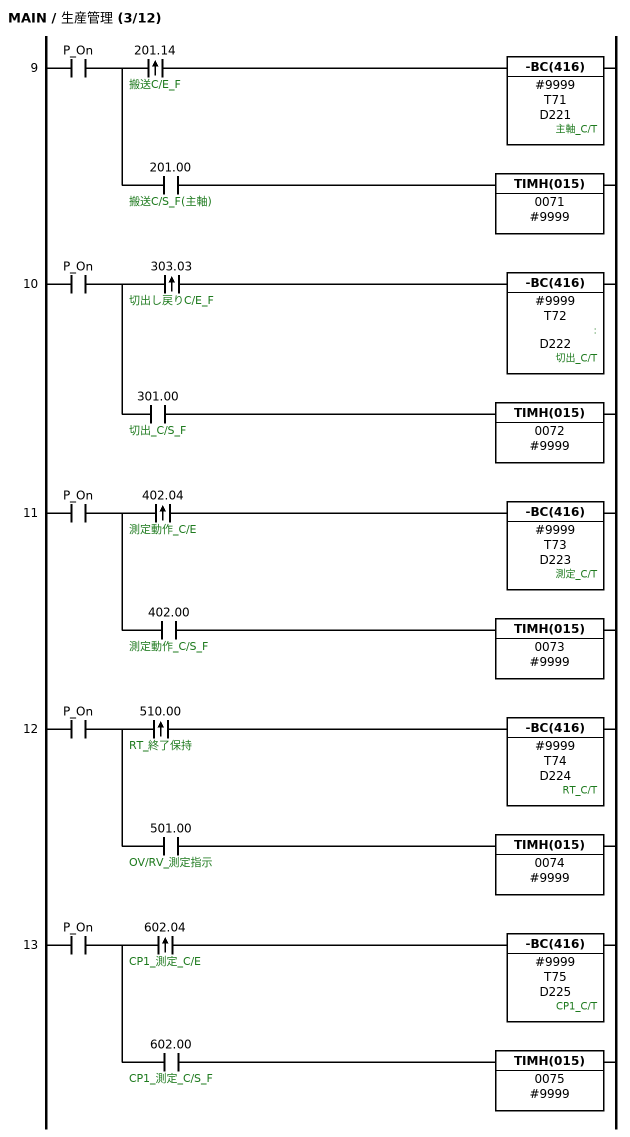
; [picture p24: MAIN / 生産管理, rungs 9-13]
; rung 9
LD P_On
OUT TR0
@AND 201.14  ; 搬送C/E_F
-BC(416) #9999 T71 D221  ; 主軸_C/T
LD TR0
AND 201.00  ; 搬送C/S_F(主軸)
TIMH(015) 0071 #9999
; rung 10
LD P_On
OUT TR0
@AND 303.03  ; 切出し戻りC/E_F
-BC(416) #9999 T72 D222  ; :, 切出_C/T
LD TR0
AND 301.00  ; 切出_C/S_F
TIMH(015) 0072 #9999
; rung 11
LD P_On
OUT TR0
@AND 402.04  ; 測定動作_C/E
-BC(416) #9999 T73 D223  ; 測定_C/T
LD TR0
AND 402.00  ; 測定動作_C/S_F
TIMH(015) 0073 #9999
; rung 12
LD P_On
OUT TR0
@AND 510.00  ; RT_終了保持
-BC(416) #9999 T74 D224  ; RT_C/T
LD TR0
AND 501.00  ; OV/RV_測定指示
TIMH(015) 0074 #9999
; rung 13
LD P_On
OUT TR0
@AND 602.04  ; CP1_測定_C/E
-BC(416) #9999 T75 D225  ; CP1_C/T
LD TR0
AND 602.00  ; CP1_測定_C/S_F
TIMH(015) 0075 #9999

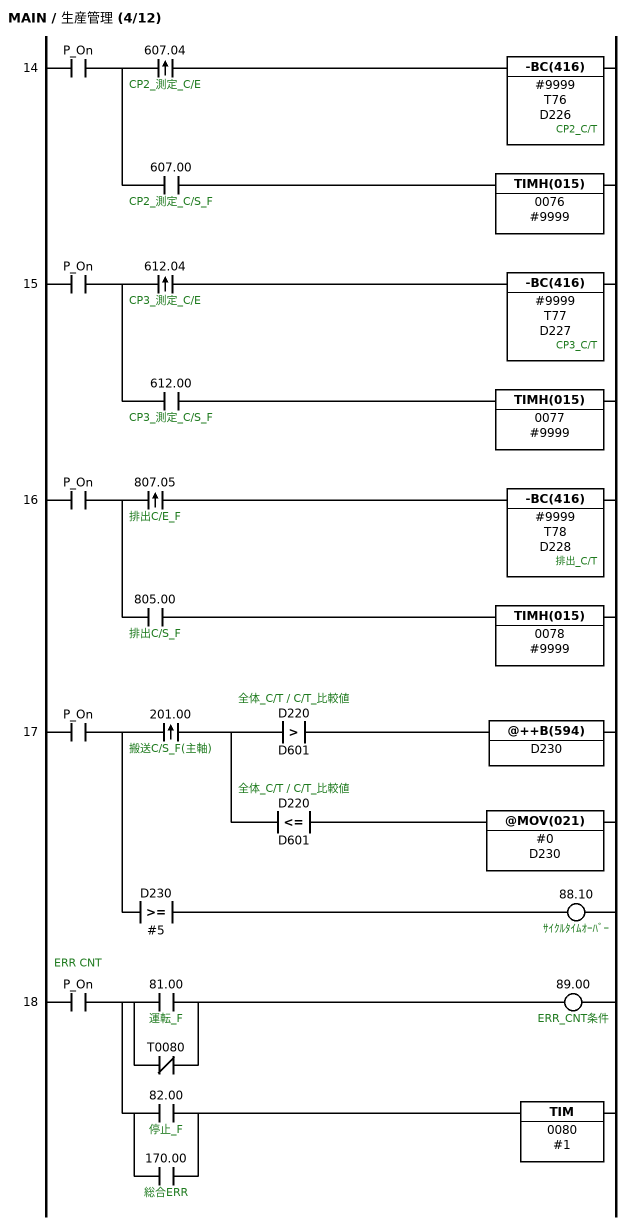
; rung 14
LD P_On
OUT TR0
@AND 607.04  ; CP2_測定_C/E
-BC(416) #9999 T76 D226  ; CP2_C/T
LD TR0
AND 607.00  ; CP2_測定_C/S_F
TIMH(015) 0076 #9999
; rung 15
LD P_On
OUT TR0
@AND 612.04  ; CP3_測定_C/E
-BC(416) #9999 T77 D227  ; CP3_C/T
LD TR0
AND 612.00  ; CP3_測定_C/S_F
TIMH(015) 0077 #9999
; rung 16
LD P_On
OUT TR0
@AND 807.05  ; 排出C/E_F
-BC(416) #9999 T78 D228  ; 排出_C/T
LD TR0
AND 805.00  ; 排出C/S_F
TIMH(015) 0078 #9999
; rung 17
LD P_On
OUT TR0
@AND 201.00  ; 搬送C/S_F(主軸)
OUT TR1
AND>(320) D220 D601  ; 全体_C/T, C/T_比較値
@++B(594) D230
LD TR1
AND<=(315) D220 D601  ; 全体_C/T, C/T_比較値
@MOV(021) #0 D230
LD TR0
AND>=(325) D230 #5
OUT 88.10  ; ｻｲｸﾙﾀｲﾑｵｰﾊﾞｰ
; rung 18: ERR CNT
LD P_On
OUT TR0
LD 81.00  ; 運転_F
ORNOT T0080
ANDLD
OUT 89.00  ; ERR_CNT条件
LD TR0
LD 82.00  ; 停止_F
OR 170.00  ; 総合ERR
ANDLD
TIM 0080 #1

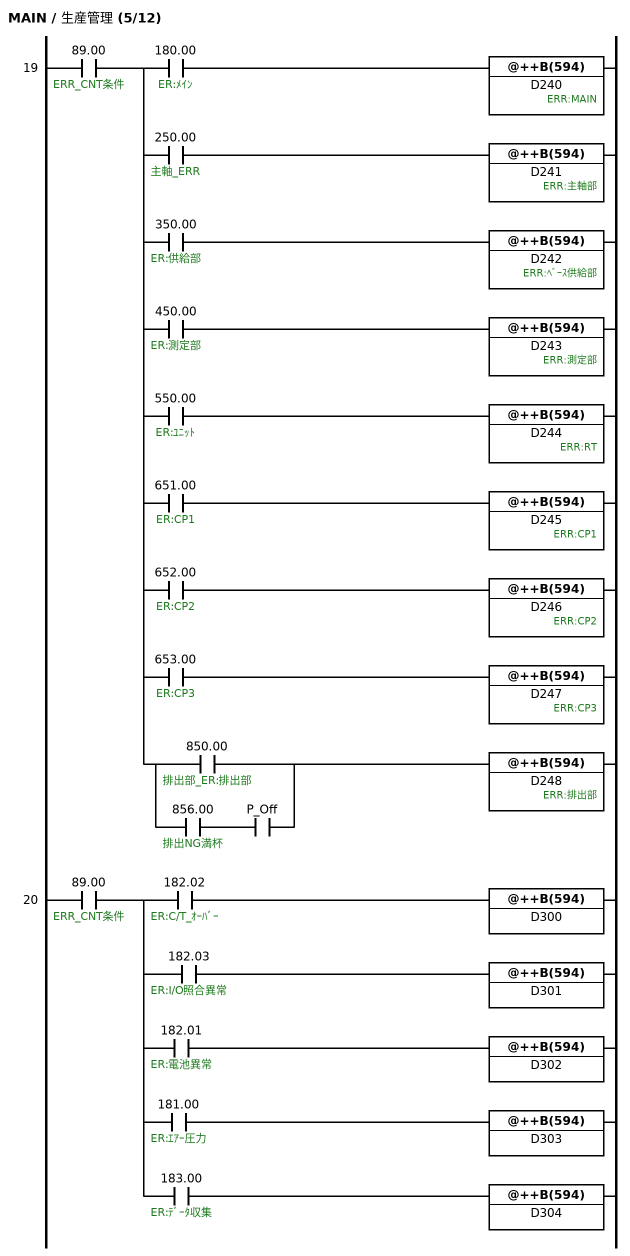
; rung 19
LD 89.00  ; ERR_CNT条件
OUT TR0
AND 180.00  ; ER:ﾒｲﾝ
@++B(594) D240  ; ERR:MAIN
LD TR0
AND 250.00  ; 主軸_ERR
@++B(594) D241  ; ERR:主軸部
LD TR0
AND 350.00  ; ER:供給部
@++B(594) D242  ; ERR:ﾍﾞｰｽ供給部
LD TR0
AND 450.00  ; ER:測定部
@++B(594) D243  ; ERR:測定部
LD TR0
AND 550.00  ; ER:ﾕﾆｯﾄ
@++B(594) D244  ; ERR:RT
LD TR0
AND 651.00  ; ER:CP1
@++B(594) D245  ; ERR:CP1
LD TR0
AND 652.00  ; ER:CP2
@++B(594) D246  ; ERR:CP2
LD TR0
AND 653.00  ; ER:CP3
@++B(594) D247  ; ERR:CP3
LD TR0
LD 850.00  ; 排出部_ER:排出部
LD 856.00  ; 排出NG満杯
AND P_Off
ORLD
ANDLD
@++B(594) D248  ; ERR:排出部
; rung 20
LD 89.00  ; ERR_CNT条件
OUT TR0
AND 182.02  ; ER:C/T_ｵｰﾊﾞｰ
@++B(594) D300
LD TR0
AND 182.03  ; ER:I/O照合異常
@++B(594) D301
LD TR0
AND 182.01  ; ER:電池異常
@++B(594) D302
LD TR0
AND 181.00  ; ER:ｴｱｰ圧力
@++B(594) D303
LD TR0
AND 183.00  ; ER:ﾃﾞｰﾀ収集
@++B(594) D304

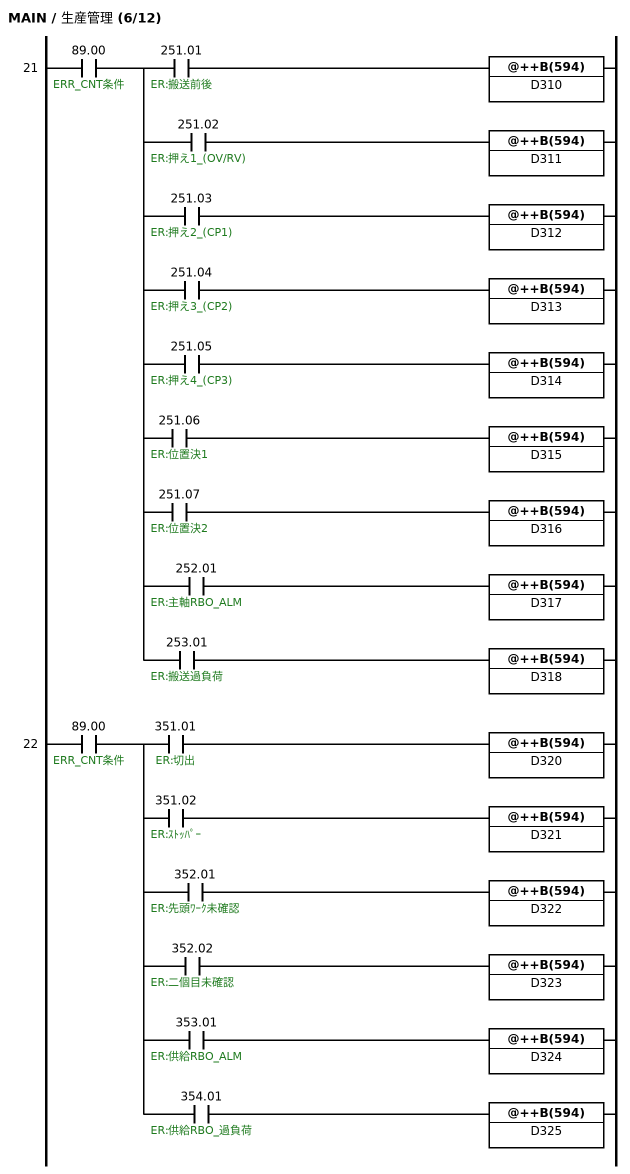
; rung 21
LD 89.00  ; ERR_CNT条件
OUT TR0
AND 251.01  ; ER:搬送前後
@++B(594) D310
LD TR0
AND 251.02  ; ER:押え1_(OV/RV)
@++B(594) D311
LD TR0
AND 251.03  ; ER:押え2_(CP1)
@++B(594) D312
LD TR0
AND 251.04  ; ER:押え3_(CP2)
@++B(594) D313
LD TR0
AND 251.05  ; ER:押え4_(CP3)
@++B(594) D314
LD TR0
AND 251.06  ; ER:位置決1
@++B(594) D315
LD TR0
AND 251.07  ; ER:位置決2
@++B(594) D316
LD TR0
AND 252.01  ; ER:主軸RBO_ALM
@++B(594) D317
LD TR0
AND 253.01  ; ER:搬送過負荷
@++B(594) D318
; rung 22
LD 89.00  ; ERR_CNT条件
OUT TR0
AND 351.01  ; ER:切出
@++B(594) D320
LD TR0
AND 351.02  ; ER:ｽﾄｯﾊﾟｰ
@++B(594) D321
LD TR0
AND 352.01  ; ER:先頭ﾜｰｸ未確認
@++B(594) D322
LD TR0
AND 352.02  ; ER:二個目未確認
@++B(594) D323
LD TR0
AND 353.01  ; ER:供給RBO_ALM
@++B(594) D324
LD TR0
AND 354.01  ; ER:供給RBO_過負荷
@++B(594) D325

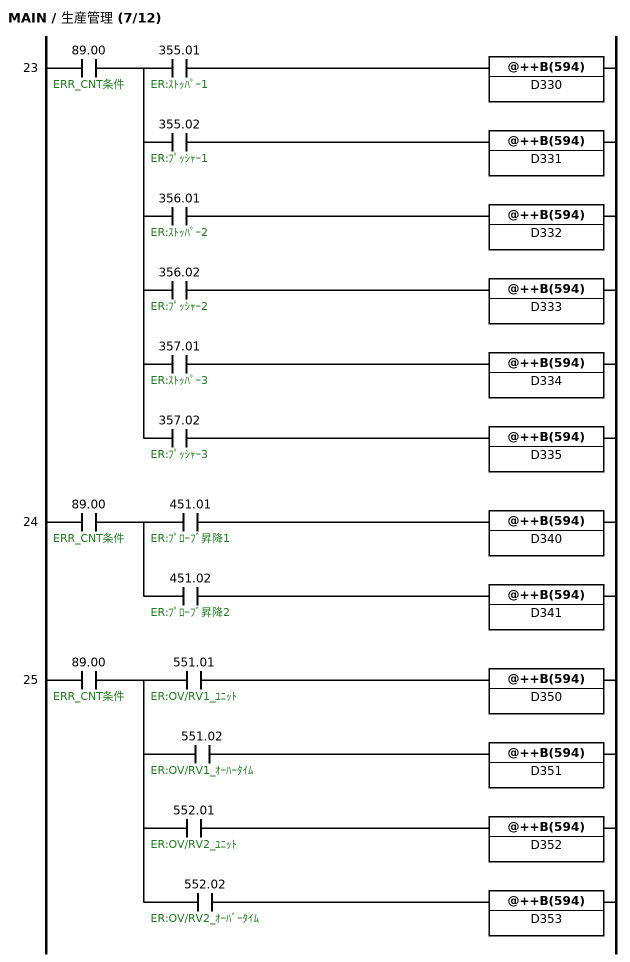
; rung 23
LD 89.00  ; ERR_CNT条件
OUT TR0
AND 355.01  ; ER:ｽﾄｯﾊﾟｰ1
@++B(594) D330
LD TR0
AND 355.02  ; ER:ﾌﾟｯｼｬｰ1
@++B(594) D331
LD TR0
AND 356.01  ; ER:ｽﾄｯﾊﾟｰ2
@++B(594) D332
LD TR0
AND 356.02  ; ER:ﾌﾟｯｼｬｰ2
@++B(594) D333
LD TR0
AND 357.01  ; ER:ｽﾄｯﾊﾟｰ3
@++B(594) D334
LD TR0
AND 357.02  ; ER:ﾌﾟｯｼｬｰ3
@++B(594) D335
; rung 24
LD 89.00  ; ERR_CNT条件
OUT TR0
AND 451.01  ; ER:ﾌﾟﾛｰﾌﾞ昇降1
@++B(594) D340
LD TR0
AND 451.02  ; ER:ﾌﾟﾛｰﾌﾞ昇降2
@++B(594) D341
; rung 25
LD 89.00  ; ERR_CNT条件
OUT TR0
AND 551.01  ; ER:OV/RV1_ﾕﾆｯﾄ
@++B(594) D350
LD TR0
AND 551.02  ; ER:OV/RV1_ｵｰﾊｰﾀｲﾑ
@++B(594) D351
LD TR0
AND 552.01  ; ER:OV/RV2_ﾕﾆｯﾄ
@++B(594) D352
LD TR0
AND 552.02  ; ER:OV/RV2_ｵｰﾊﾞｰﾀｲﾑ
@++B(594) D353

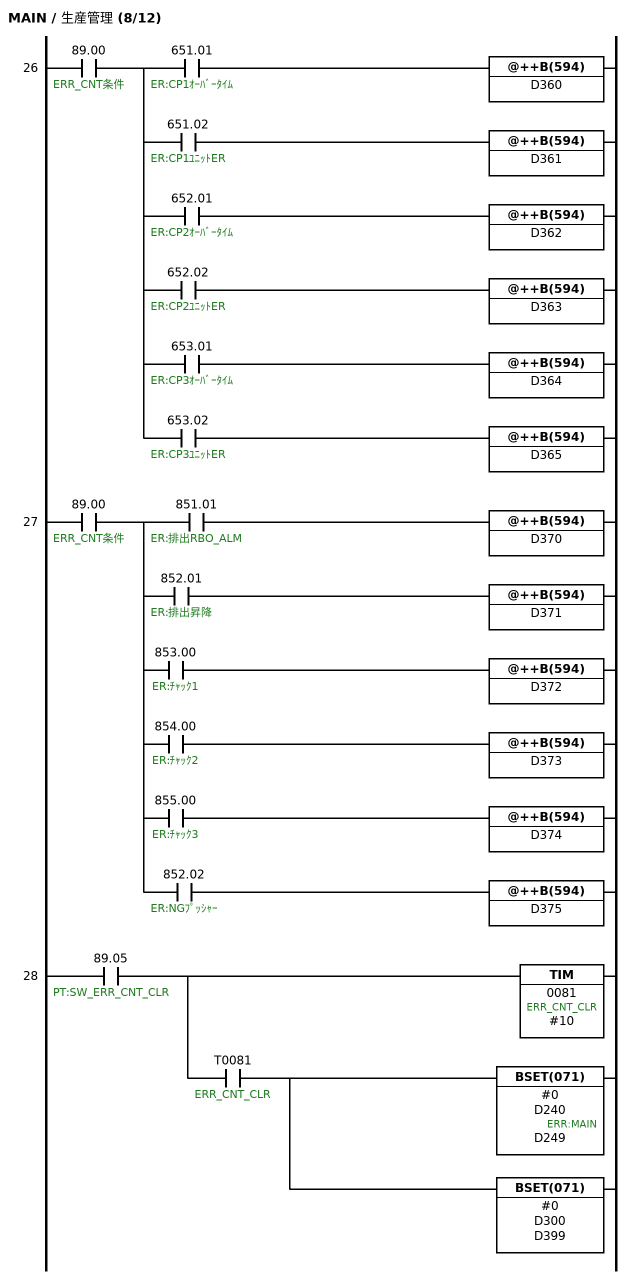
; rung 26
LD 89.00  ; ERR_CNT条件
OUT TR0
AND 651.01  ; ER:CP1ｵｰﾊﾞｰﾀｲﾑ
@++B(594) D360
LD TR0
AND 651.02  ; ER:CP1ﾕﾆｯﾄER
@++B(594) D361
LD TR0
AND 652.01  ; ER:CP2ｵｰﾊﾞｰﾀｲﾑ
@++B(594) D362
LD TR0
AND 652.02  ; ER:CP2ﾕﾆｯﾄER
@++B(594) D363
LD TR0
AND 653.01  ; ER:CP3ｵｰﾊﾞｰﾀｲﾑ
@++B(594) D364
LD TR0
AND 653.02  ; ER:CP3ﾕﾆｯﾄER
@++B(594) D365
; rung 27
LD 89.00  ; ERR_CNT条件
OUT TR0
AND 851.01  ; ER:排出RBO_ALM
@++B(594) D370
LD TR0
AND 852.01  ; ER:排出昇降
@++B(594) D371
LD TR0
AND 853.00  ; ER:ﾁｬｯｸ1
@++B(594) D372
LD TR0
AND 854.00  ; ER:ﾁｬｯｸ2
@++B(594) D373
LD TR0
AND 855.00  ; ER:ﾁｬｯｸ3
@++B(594) D374
LD TR0
AND 852.02  ; ER:NGﾌﾟｯｼｬｰ
@++B(594) D375
; rung 28
LD 89.05  ; PT:SW_ERR_CNT_CLR
TIM 0081 #10  ; ERR_CNT_CLR
AND T0081  ; ERR_CNT_CLR
BSET(071) #0 D240 D249  ; ERR:MAIN
BSET(071) #0 D300 D399

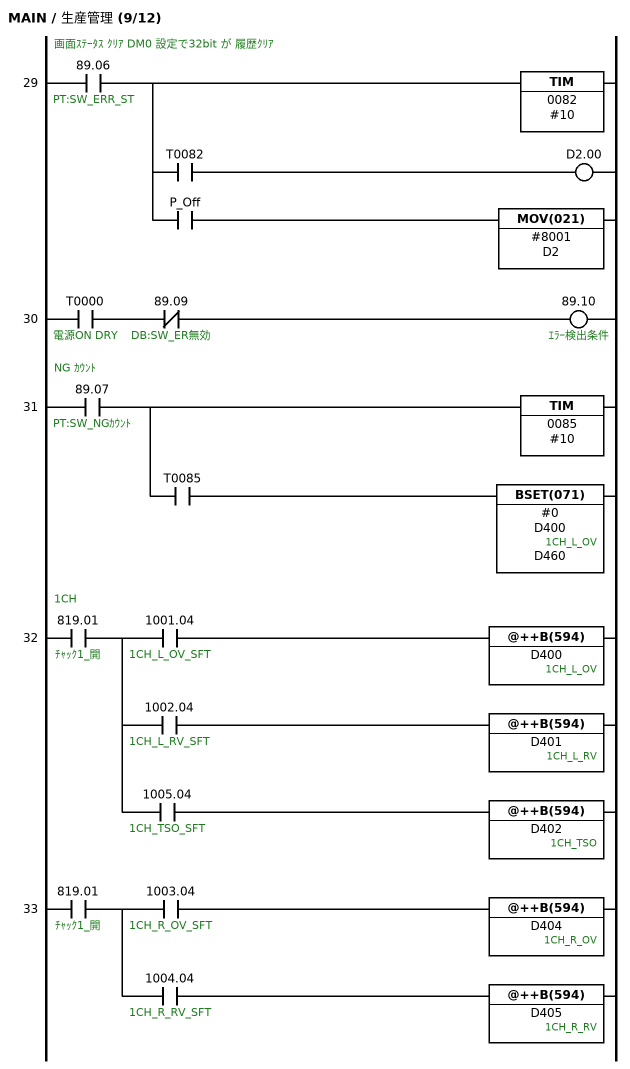
; rung 29: 画面ｽﾃｰﾀｽ ｸﾘｱ DM0 設定で32bit が 履歴ｸﾘｱ
LD 89.06  ; PT:SW_ERR_ST
OUT TR0
TIM 0082 #10
AND T0082
OUT D2.00
LD TR0
AND P_Off
MOV(021) #8001 D2
; rung 30
LD T0000  ; 電源ON DRY
ANDNOT 89.09  ; DB:SW_ER無効
OUT 89.10  ; ｴﾗｰ検出条件
; rung 31: NG ｶｳﾝﾄ
LD 89.07  ; PT:SW_NGｶｳﾝﾄ
TIM 0085 #10
AND T0085
BSET(071) #0 D400 D460  ; 1CH_L_OV
; rung 32: 1CH
LD 819.01  ; ﾁｬｯｸ1_開
OUT TR0
AND 1001.04  ; 1CH_L_OV_SFT
@++B(594) D400  ; 1CH_L_OV
LD TR0
AND 1002.04  ; 1CH_L_RV_SFT
@++B(594) D401  ; 1CH_L_RV
LD TR0
AND 1005.04  ; 1CH_TSO_SFT
@++B(594) D402  ; 1CH_TSO
; rung 33
LD 819.01  ; ﾁｬｯｸ1_開
OUT TR0
AND 1003.04  ; 1CH_R_OV_SFT
@++B(594) D404  ; 1CH_R_OV
LD TR0
AND 1004.04  ; 1CH_R_RV_SFT
@++B(594) D405  ; 1CH_R_RV

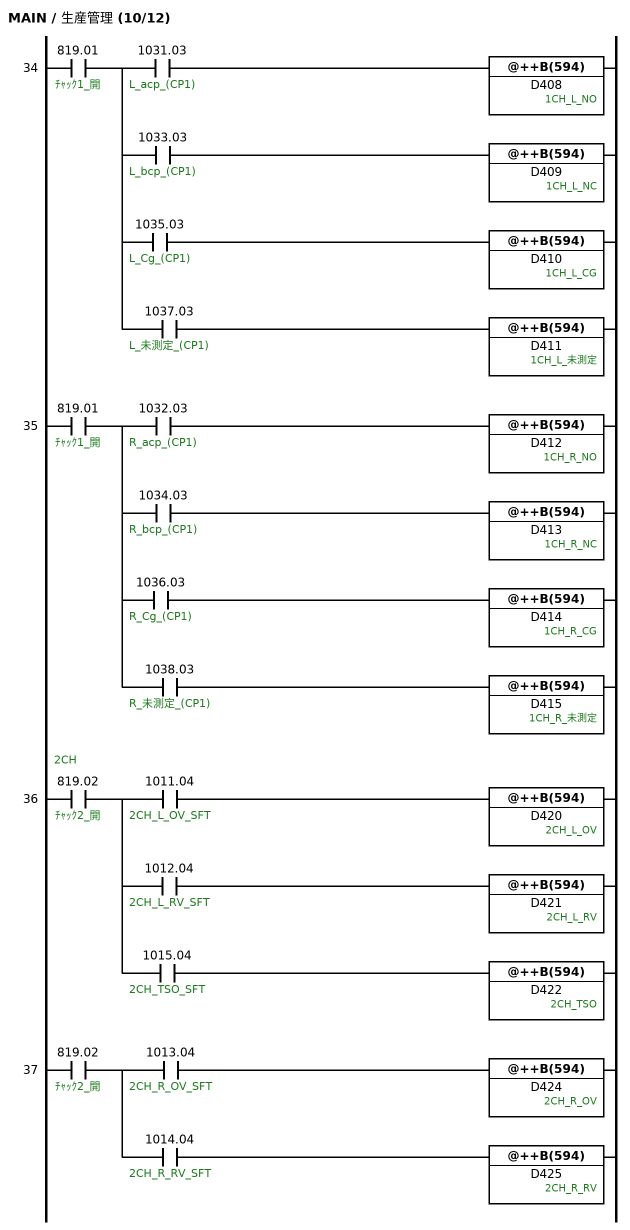
; rung 34
LD 819.01  ; ﾁｬｯｸ1_開
OUT TR0
AND 1031.03  ; L_acp_(CP1)
@++B(594) D408  ; 1CH_L_NO
LD TR0
AND 1033.03  ; L_bcp_(CP1)
@++B(594) D409  ; 1CH_L_NC
LD TR0
AND 1035.03  ; L_Cg_(CP1)
@++B(594) D410  ; 1CH_L_CG
LD TR0
AND 1037.03  ; L_未測定_(CP1)
@++B(594) D411  ; 1CH_L_未測定
; rung 35
LD 819.01  ; ﾁｬｯｸ1_開
OUT TR0
AND 1032.03  ; R_acp_(CP1)
@++B(594) D412  ; 1CH_R_NO
LD TR0
AND 1034.03  ; R_bcp_(CP1)
@++B(594) D413  ; 1CH_R_NC
LD TR0
AND 1036.03  ; R_Cg_(CP1)
@++B(594) D414  ; 1CH_R_CG
LD TR0
AND 1038.03  ; R_未測定_(CP1)
@++B(594) D415  ; 1CH_R_未測定
; rung 36: 2CH
LD 819.02  ; ﾁｬｯｸ2_開
OUT TR0
AND 1011.04  ; 2CH_L_OV_SFT
@++B(594) D420  ; 2CH_L_OV
LD TR0
AND 1012.04  ; 2CH_L_RV_SFT
@++B(594) D421  ; 2CH_L_RV
LD TR0
AND 1015.04  ; 2CH_TSO_SFT
@++B(594) D422  ; 2CH_TSO
; rung 37
LD 819.02  ; ﾁｬｯｸ2_開
OUT TR0
AND 1013.04  ; 2CH_R_OV_SFT
@++B(594) D424  ; 2CH_R_OV
LD TR0
AND 1014.04  ; 2CH_R_RV_SFT
@++B(594) D425  ; 2CH_R_RV

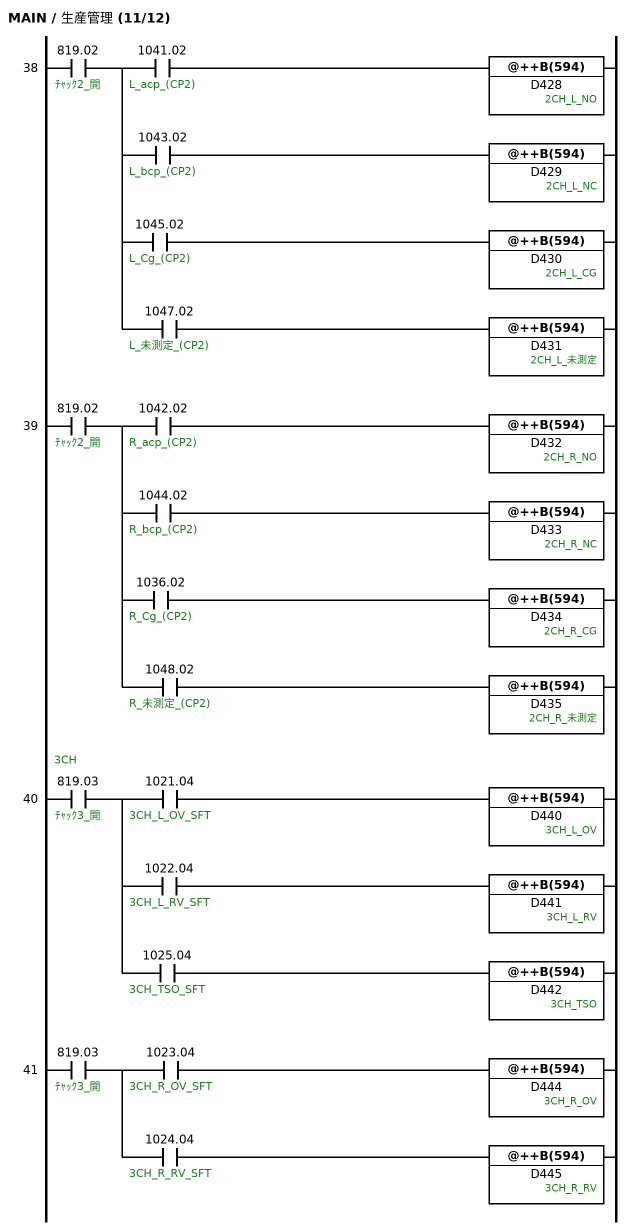
; rung 38
LD 819.02  ; ﾁｬｯｸ2_開
OUT TR0
AND 1041.02  ; L_acp_(CP2)
@++B(594) D428  ; 2CH_L_NO
LD TR0
AND 1043.02  ; L_bcp_(CP2)
@++B(594) D429  ; 2CH_L_NC
LD TR0
AND 1045.02  ; L_Cg_(CP2)
@++B(594) D430  ; 2CH_L_CG
LD TR0
AND 1047.02  ; L_未測定_(CP2)
@++B(594) D431  ; 2CH_L_未測定
; rung 39
LD 819.02  ; ﾁｬｯｸ2_開
OUT TR0
AND 1042.02  ; R_acp_(CP2)
@++B(594) D432  ; 2CH_R_NO
LD TR0
AND 1044.02  ; R_bcp_(CP2)
@++B(594) D433  ; 2CH_R_NC
LD TR0
AND 1036.02  ; R_Cg_(CP2)
@++B(594) D434  ; 2CH_R_CG
LD TR0
AND 1048.02  ; R_未測定_(CP2)
@++B(594) D435  ; 2CH_R_未測定
; rung 40: 3CH
LD 819.03  ; ﾁｬｯｸ3_開
OUT TR0
AND 1021.04  ; 3CH_L_OV_SFT
@++B(594) D440  ; 3CH_L_OV
LD TR0
AND 1022.04  ; 3CH_L_RV_SFT
@++B(594) D441  ; 3CH_L_RV
LD TR0
AND 1025.04  ; 3CH_TSO_SFT
@++B(594) D442  ; 3CH_TSO
; rung 41
LD 819.03  ; ﾁｬｯｸ3_開
OUT TR0
AND 1023.04  ; 3CH_R_OV_SFT
@++B(594) D444  ; 3CH_R_OV
LD TR0
AND 1024.04  ; 3CH_R_RV_SFT
@++B(594) D445  ; 3CH_R_RV

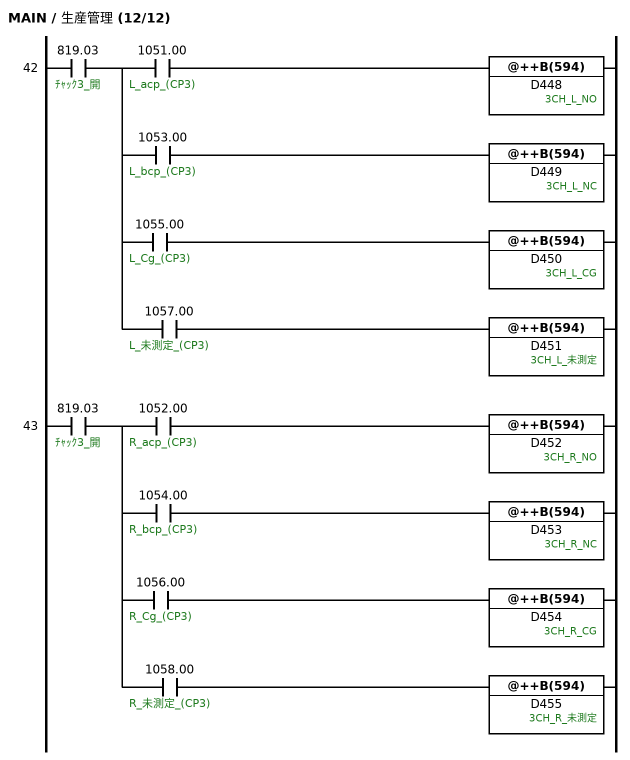
; rung 42
LD 819.03  ; ﾁｬｯｸ3_開
OUT TR0
AND 1051.00  ; L_acp_(CP3)
@++B(594) D448  ; 3CH_L_NO
LD TR0
AND 1053.00  ; L_bcp_(CP3)
@++B(594) D449  ; 3CH_L_NC
LD TR0
AND 1055.00  ; L_Cg_(CP3)
@++B(594) D450  ; 3CH_L_CG
LD TR0
AND 1057.00  ; L_未測定_(CP3)
@++B(594) D451  ; 3CH_L_未測定
; rung 43
LD 819.03  ; ﾁｬｯｸ3_開
OUT TR0
AND 1052.00  ; R_acp_(CP3)
@++B(594) D452  ; 3CH_R_NO
LD TR0
AND 1054.00  ; R_bcp_(CP3)
@++B(594) D453  ; 3CH_R_NC
LD TR0
AND 1056.00  ; R_Cg_(CP3)
@++B(594) D454  ; 3CH_R_CG
LD TR0
AND 1058.00  ; R_未測定_(CP3)
@++B(594) D455  ; 3CH_R_未測定

### Section ERR

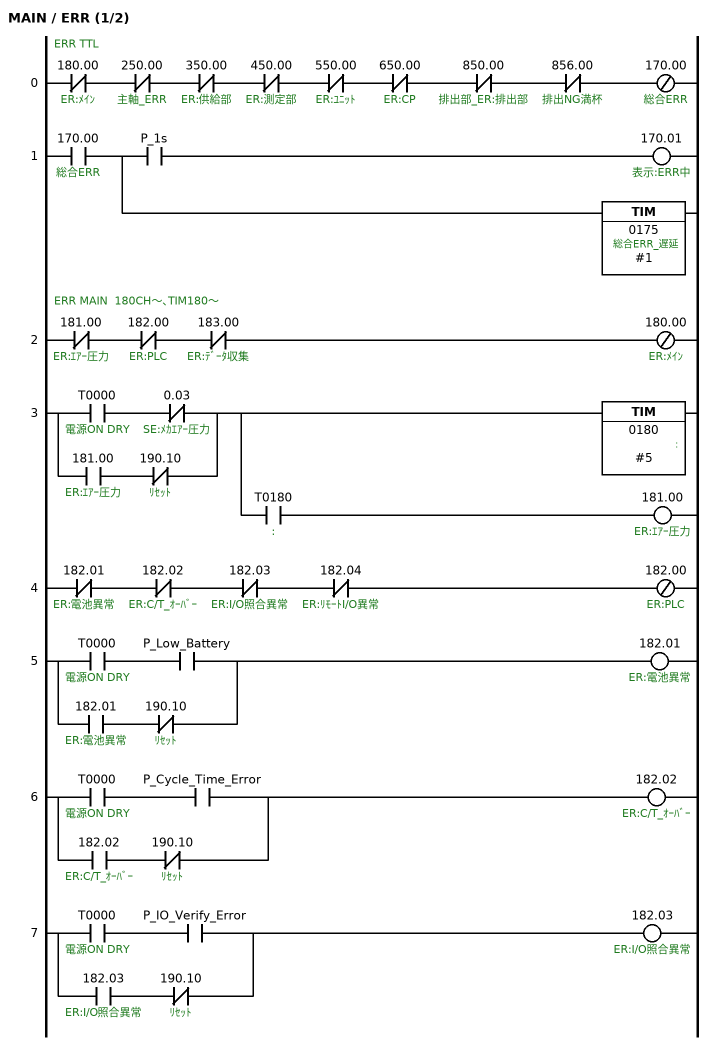
; rung 0: ERR TTL
LDNOT 180.00  ; ER:ﾒｲﾝ
ANDNOT 250.00  ; 主軸_ERR
ANDNOT 350.00  ; ER:供給部
ANDNOT 450.00  ; ER:測定部
ANDNOT 550.00  ; ER:ﾕﾆｯﾄ
ANDNOT 650.00  ; ER:CP
ANDNOT 850.00  ; 排出部_ER:排出部
ANDNOT 856.00  ; 排出NG満杯
OUTNOT 170.00  ; 総合ERR
; rung 1
LD 170.00  ; 総合ERR
OUT TR0
AND P_1s
OUT 170.01  ; 表示:ERR中
LD TR0
TIM 0175 #1  ; 総合ERR_遅延
; rung 2: ERR MAIN  180CH～､TIM180～
LDNOT 181.00  ; ER:ｴｱｰ圧力
ANDNOT 182.00  ; ER:PLC
ANDNOT 183.00  ; ER:ﾃﾞｰﾀ収集
OUTNOT 180.00  ; ER:ﾒｲﾝ
; rung 3
LD T0000  ; 電源ON DRY
ANDNOT 0.03  ; SE:ﾒｶｴｱｰ圧力
LD 181.00  ; ER:ｴｱｰ圧力
ANDNOT 190.10  ; ﾘｾｯﾄ
ORLD
TIM 0180 #5  ; :
AND T0180  ; :
OUT 181.00  ; ER:ｴｱｰ圧力
; rung 4
LDNOT 182.01  ; ER:電池異常
ANDNOT 182.02  ; ER:C/T_ｵｰﾊﾞｰ
ANDNOT 182.03  ; ER:I/O照合異常
ANDNOT 182.04  ; ER:ﾘﾓｰﾄI/O異常
OUTNOT 182.00  ; ER:PLC
; rung 5
LD T0000  ; 電源ON DRY
AND P_Low_Battery
LD 182.01  ; ER:電池異常
ANDNOT 190.10  ; ﾘｾｯﾄ
ORLD
OUT 182.01  ; ER:電池異常
; rung 6
LD T0000  ; 電源ON DRY
AND P_Cycle_Time_Error
LD 182.02  ; ER:C/T_ｵｰﾊﾞｰ
ANDNOT 190.10  ; ﾘｾｯﾄ
ORLD
OUT 182.02  ; ER:C/T_ｵｰﾊﾞｰ
; rung 7
LD T0000  ; 電源ON DRY
AND P_IO_Verify_Error
LD 182.03  ; ER:I/O照合異常
ANDNOT 190.10  ; ﾘｾｯﾄ
ORLD
OUT 182.03  ; ER:I/O照合異常

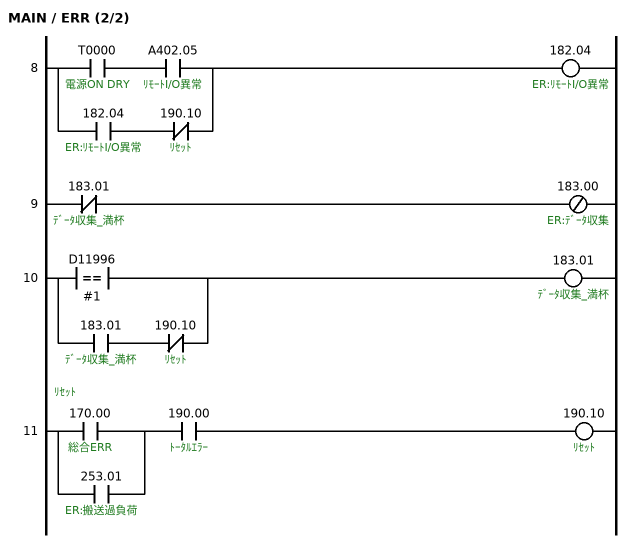
; rung 8
LD T0000  ; 電源ON DRY
AND A402.05  ; ﾘﾓｰﾄI/O異常
LD 182.04  ; ER:ﾘﾓｰﾄI/O異常
ANDNOT 190.10  ; ﾘｾｯﾄ
ORLD
OUT 182.04  ; ER:ﾘﾓｰﾄI/O異常
; rung 9
LDNOT 183.01  ; ﾃﾞｰﾀ収集_満杯
OUTNOT 183.00  ; ER:ﾃﾞｰﾀ収集
; rung 10
LD=(300) D11996 #1
LD 183.01  ; ﾃﾞｰﾀ収集_満杯
ANDNOT 190.10  ; ﾘｾｯﾄ
ORLD
OUT 183.01  ; ﾃﾞｰﾀ収集_満杯
; rung 11: ﾘｾｯﾄ
LD 170.00  ; 総合ERR
OR 253.01  ; ER:搬送過負荷
AND 190.00  ; ﾄｰﾀﾙｴﾗｰ
OUT 190.10  ; ﾘｾｯﾄ

### Section END
; rung 0
END(001)

## Program MANU (cyclic task 1)

### Section IL

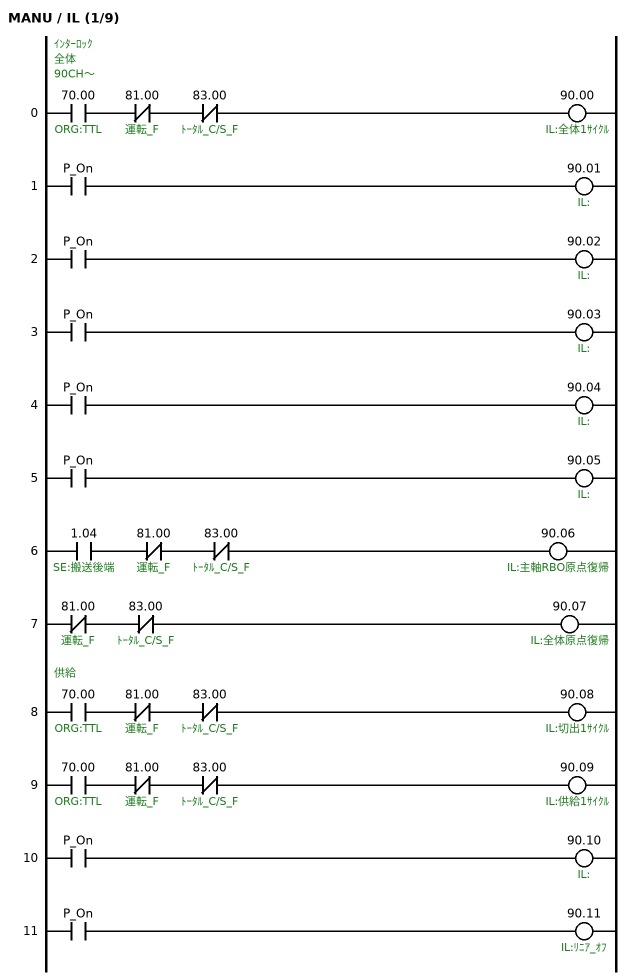
; rung 0: ｲﾝﾀｰﾛｯｸ / 全体 / 90CH～
LD 70.00  ; ORG:TTL
ANDNOT 81.00  ; 運転_F
ANDNOT 83.00  ; ﾄｰﾀﾙ_C/S_F
OUT 90.00  ; IL:全体1ｻｲｸﾙ
; rung 1
LD P_On
OUT 90.01  ; IL:
; rung 2
LD P_On
OUT 90.02  ; IL:
; rung 3
LD P_On
OUT 90.03  ; IL:
; rung 4
LD P_On
OUT 90.04  ; IL:
; rung 5
LD P_On
OUT 90.05  ; IL:
; rung 6
LD 1.04  ; SE:搬送後端
ANDNOT 81.00  ; 運転_F
ANDNOT 83.00  ; ﾄｰﾀﾙ_C/S_F
OUT 90.06  ; IL:主軸RBO原点復帰
; rung 7
LDNOT 81.00  ; 運転_F
ANDNOT 83.00  ; ﾄｰﾀﾙ_C/S_F
OUT 90.07  ; IL:全体原点復帰
; rung 8: 供給
LD 70.00  ; ORG:TTL
ANDNOT 81.00  ; 運転_F
ANDNOT 83.00  ; ﾄｰﾀﾙ_C/S_F
OUT 90.08  ; IL:切出1ｻｲｸﾙ
; rung 9
LD 70.00  ; ORG:TTL
ANDNOT 81.00  ; 運転_F
ANDNOT 83.00  ; ﾄｰﾀﾙ_C/S_F
OUT 90.09  ; IL:供給1ｻｲｸﾙ
; rung 10
LD P_On
OUT 90.10  ; IL:
; rung 11
LD P_On
OUT 90.11  ; IL:ﾘﾆｱ_ｵﾌ

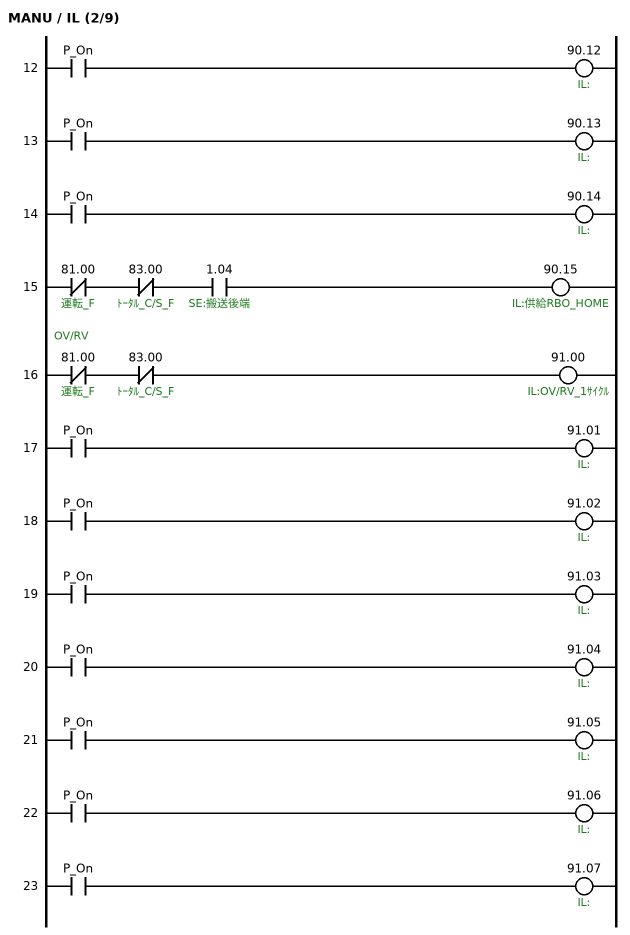
; rung 12
LD P_On
OUT 90.12  ; IL:
; rung 13
LD P_On
OUT 90.13  ; IL:
; rung 14
LD P_On
OUT 90.14  ; IL:
; rung 15
LDNOT 81.00  ; 運転_F
ANDNOT 83.00  ; ﾄｰﾀﾙ_C/S_F
AND 1.04  ; SE:搬送後端
OUT 90.15  ; IL:供給RBO_HOME
; rung 16: OV/RV
LDNOT 81.00  ; 運転_F
ANDNOT 83.00  ; ﾄｰﾀﾙ_C/S_F
OUT 91.00  ; IL:OV/RV_1ｻｲｸﾙ
; rung 17
LD P_On
OUT 91.01  ; IL:
; rung 18
LD P_On
OUT 91.02  ; IL:
; rung 19
LD P_On
OUT 91.03  ; IL:
; rung 20
LD P_On
OUT 91.04  ; IL:
; rung 21
LD P_On
OUT 91.05  ; IL:
; rung 22
LD P_On
OUT 91.06  ; IL:
; rung 23
LD P_On
OUT 91.07  ; IL:

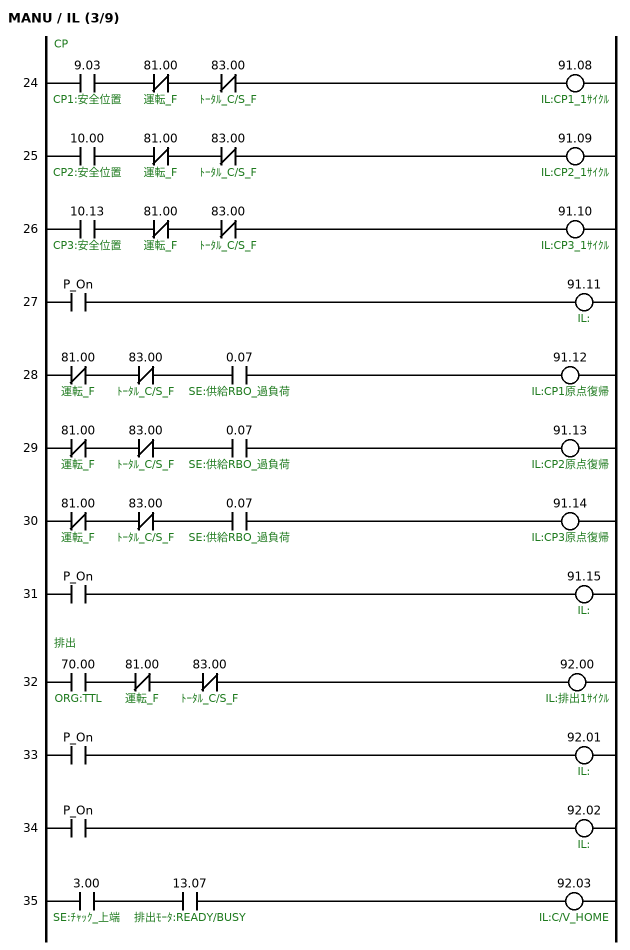
; rung 24: CP
LD 9.03  ; CP1:安全位置
ANDNOT 81.00  ; 運転_F
ANDNOT 83.00  ; ﾄｰﾀﾙ_C/S_F
OUT 91.08  ; IL:CP1_1ｻｲｸﾙ
; rung 25
LD 10.00  ; CP2:安全位置
ANDNOT 81.00  ; 運転_F
ANDNOT 83.00  ; ﾄｰﾀﾙ_C/S_F
OUT 91.09  ; IL:CP2_1ｻｲｸﾙ
; rung 26
LD 10.13  ; CP3:安全位置
ANDNOT 81.00  ; 運転_F
ANDNOT 83.00  ; ﾄｰﾀﾙ_C/S_F
OUT 91.10  ; IL:CP3_1ｻｲｸﾙ
; rung 27
LD P_On
OUT 91.11  ; IL:
; rung 28
LDNOT 81.00  ; 運転_F
ANDNOT 83.00  ; ﾄｰﾀﾙ_C/S_F
AND 0.07  ; SE:供給RBO_過負荷
OUT 91.12  ; IL:CP1原点復帰
; rung 29
LDNOT 81.00  ; 運転_F
ANDNOT 83.00  ; ﾄｰﾀﾙ_C/S_F
AND 0.07  ; SE:供給RBO_過負荷
OUT 91.13  ; IL:CP2原点復帰
; rung 30
LDNOT 81.00  ; 運転_F
ANDNOT 83.00  ; ﾄｰﾀﾙ_C/S_F
AND 0.07  ; SE:供給RBO_過負荷
OUT 91.14  ; IL:CP3原点復帰
; rung 31
LD P_On
OUT 91.15  ; IL:
; rung 32: 排出
LD 70.00  ; ORG:TTL
ANDNOT 81.00  ; 運転_F
ANDNOT 83.00  ; ﾄｰﾀﾙ_C/S_F
OUT 92.00  ; IL:排出1ｻｲｸﾙ
; rung 33
LD P_On
OUT 92.01  ; IL:
; rung 34
LD P_On
OUT 92.02  ; IL:
; rung 35
LD 3.00  ; SE:ﾁｬｯｸ_上端
AND 13.07  ; 排出ﾓｰﾀ:READY/BUSY
OUT 92.03  ; IL:C/V_HOME

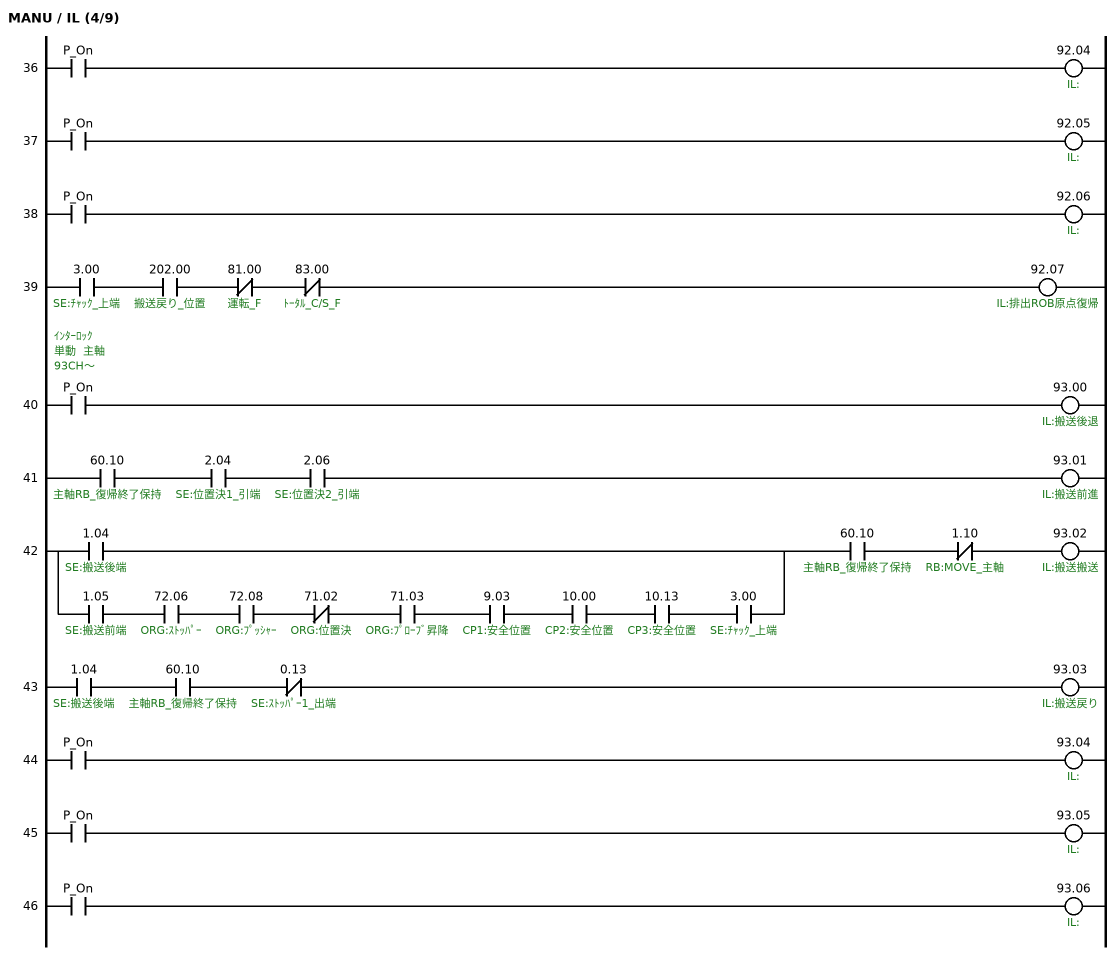
; rung 36
LD P_On
OUT 92.04  ; IL:
; rung 37
LD P_On
OUT 92.05  ; IL:
; rung 38
LD P_On
OUT 92.06  ; IL:
; rung 39
LD 3.00  ; SE:ﾁｬｯｸ_上端
AND 202.00  ; 搬送戻り_位置
ANDNOT 81.00  ; 運転_F
ANDNOT 83.00  ; ﾄｰﾀﾙ_C/S_F
OUT 92.07  ; IL:排出ROB原点復帰
; rung 40: ｲﾝﾀｰﾛｯｸ / 単動  主軸 / 93CH～
LD P_On
OUT 93.00  ; IL:搬送後退
; rung 41
LD 60.10  ; 主軸RB_復帰終了保持
AND 2.04  ; SE:位置決1_引端
AND 2.06  ; SE:位置決2_引端
OUT 93.01  ; IL:搬送前進
; rung 42
LD 1.04  ; SE:搬送後端
LD 1.05  ; SE:搬送前端
AND 72.06  ; ORG:ｽﾄｯﾊﾟｰ
AND 72.08  ; ORG:ﾌﾟｯｼｬｰ
ANDNOT 71.02  ; ORG:位置決
AND 71.03  ; ORG:ﾌﾟﾛｰﾌﾞ昇降
AND 9.03  ; CP1:安全位置
AND 10.00  ; CP2:安全位置
AND 10.13  ; CP3:安全位置
AND 3.00  ; SE:ﾁｬｯｸ_上端
ORLD
AND 60.10  ; 主軸RB_復帰終了保持
ANDNOT 1.10  ; RB:MOVE_主軸
OUT 93.02  ; IL:搬送搬送
; rung 43
LD 1.04  ; SE:搬送後端
AND 60.10  ; 主軸RB_復帰終了保持
ANDNOT 0.13  ; SE:ｽﾄｯﾊﾟｰ1_出端
OUT 93.03  ; IL:搬送戻り
; rung 44
LD P_On
OUT 93.04  ; IL:
; rung 45
LD P_On
OUT 93.05  ; IL:
; rung 46
LD P_On
OUT 93.06  ; IL:

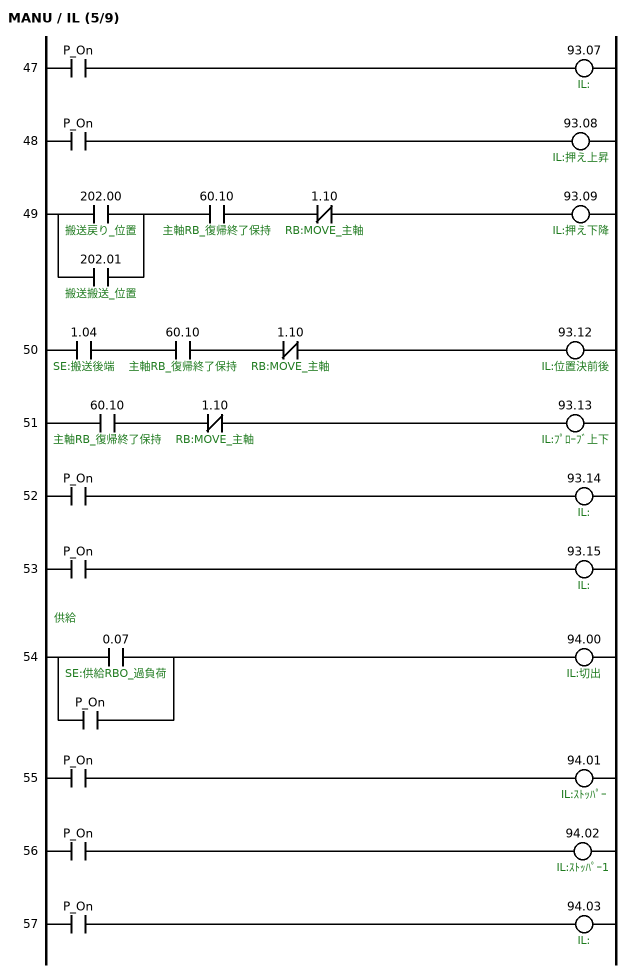
; rung 47
LD P_On
OUT 93.07  ; IL:
; rung 48
LD P_On
OUT 93.08  ; IL:押え上昇
; rung 49
LD 202.00  ; 搬送戻り_位置
OR 202.01  ; 搬送搬送_位置
AND 60.10  ; 主軸RB_復帰終了保持
ANDNOT 1.10  ; RB:MOVE_主軸
OUT 93.09  ; IL:押え下降
; rung 50
LD 1.04  ; SE:搬送後端
AND 60.10  ; 主軸RB_復帰終了保持
ANDNOT 1.10  ; RB:MOVE_主軸
OUT 93.12  ; IL:位置決前後
; rung 51
LD 60.10  ; 主軸RB_復帰終了保持
ANDNOT 1.10  ; RB:MOVE_主軸
OUT 93.13  ; IL:ﾌﾟﾛｰﾌﾞ上下
; rung 52
LD P_On
OUT 93.14  ; IL:
; rung 53
LD P_On
OUT 93.15  ; IL:
; rung 54: 供給
LD 0.07  ; SE:供給RBO_過負荷
OR P_On
OUT 94.00  ; IL:切出
; rung 55
LD P_On
OUT 94.01  ; IL:ｽﾄｯﾊﾟｰ
; rung 56
LD P_On
OUT 94.02  ; IL:ｽﾄｯﾊﾟｰ1
; rung 57
LD P_On
OUT 94.03  ; IL:

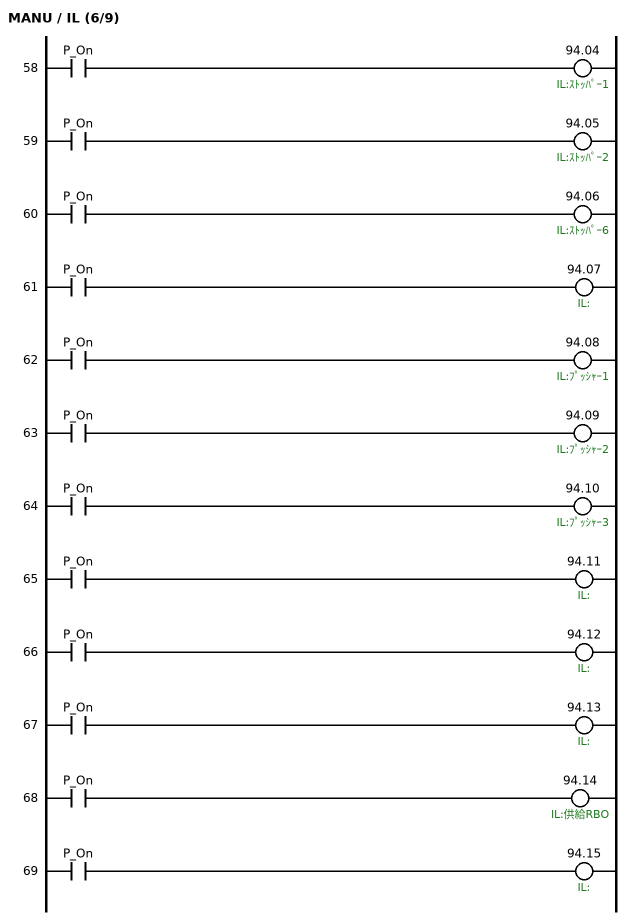
; rung 58
LD P_On
OUT 94.04  ; IL:ｽﾄｯﾊﾟｰ1
; rung 59
LD P_On
OUT 94.05  ; IL:ｽﾄｯﾊﾟｰ2
; rung 60
LD P_On
OUT 94.06  ; IL:ｽﾄｯﾊﾟｰ6
; rung 61
LD P_On
OUT 94.07  ; IL:
; rung 62
LD P_On
OUT 94.08  ; IL:ﾌﾟｯｼｬｰ1
; rung 63
LD P_On
OUT 94.09  ; IL:ﾌﾟｯｼｬｰ2
; rung 64
LD P_On
OUT 94.10  ; IL:ﾌﾟｯｼｬｰ3
; rung 65
LD P_On
OUT 94.11  ; IL:
; rung 66
LD P_On
OUT 94.12  ; IL:
; rung 67
LD P_On
OUT 94.13  ; IL:
; rung 68
LD P_On
OUT 94.14  ; IL:供給RBO
; rung 69
LD P_On
OUT 94.15  ; IL:

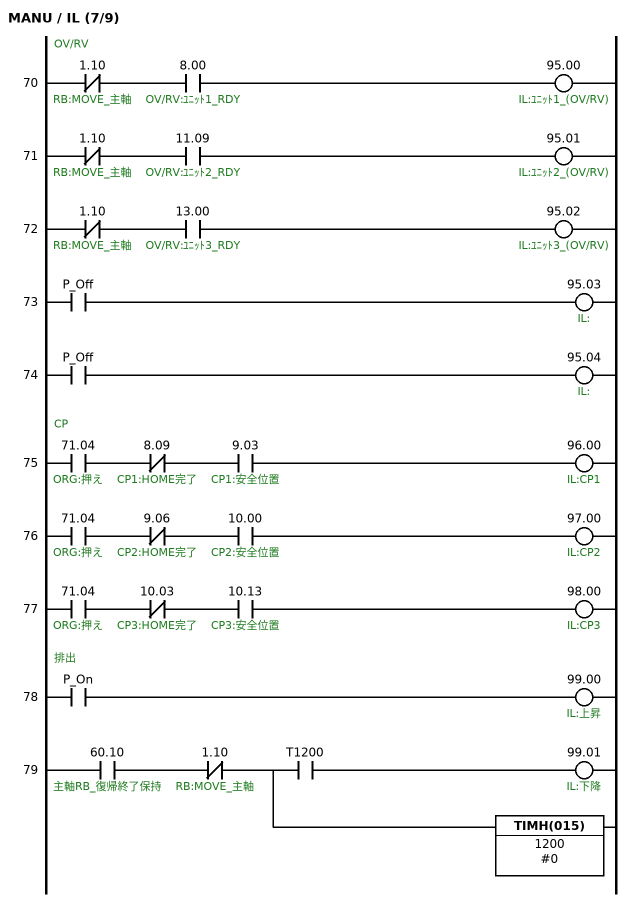
; rung 70: OV/RV
LDNOT 1.10  ; RB:MOVE_主軸
AND 8.00  ; OV/RV:ﾕﾆｯﾄ1_RDY
OUT 95.00  ; IL:ﾕﾆｯﾄ1_(OV/RV)
; rung 71
LDNOT 1.10  ; RB:MOVE_主軸
AND 11.09  ; OV/RV:ﾕﾆｯﾄ2_RDY
OUT 95.01  ; IL:ﾕﾆｯﾄ2_(OV/RV)
; rung 72
LDNOT 1.10  ; RB:MOVE_主軸
AND 13.00  ; OV/RV:ﾕﾆｯﾄ3_RDY
OUT 95.02  ; IL:ﾕﾆｯﾄ3_(OV/RV)
; rung 73
LD P_Off
OUT 95.03  ; IL:
; rung 74
LD P_Off
OUT 95.04  ; IL:
; rung 75: CP
LD 71.04  ; ORG:押え
ANDNOT 8.09  ; CP1:HOME完了
AND 9.03  ; CP1:安全位置
OUT 96.00  ; IL:CP1
; rung 76
LD 71.04  ; ORG:押え
ANDNOT 9.06  ; CP2:HOME完了
AND 10.00  ; CP2:安全位置
OUT 97.00  ; IL:CP2
; rung 77
LD 71.04  ; ORG:押え
ANDNOT 10.03  ; CP3:HOME完了
AND 10.13  ; CP3:安全位置
OUT 98.00  ; IL:CP3
; rung 78: 排出
LD P_On
OUT 99.00  ; IL:上昇
; rung 79
LD 60.10  ; 主軸RB_復帰終了保持
ANDNOT 1.10  ; RB:MOVE_主軸
OUT TR0
AND T1200
OUT 99.01  ; IL:下降
LD TR0
TIMH(015) 1200 #0

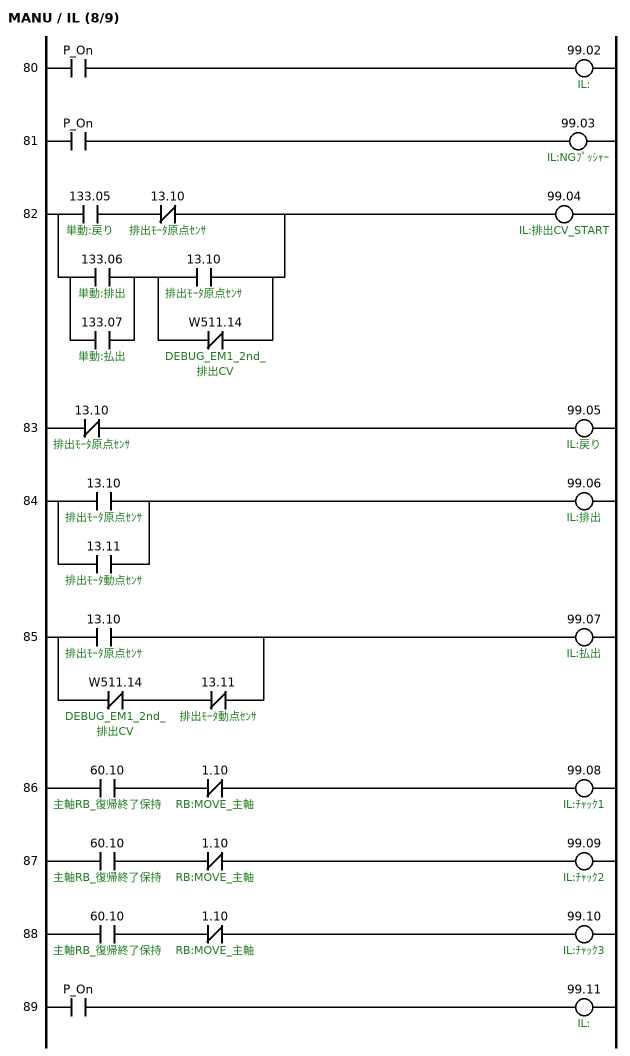
; rung 80
LD P_On
OUT 99.02  ; IL:
; rung 81
LD P_On
OUT 99.03  ; IL:NGﾌﾟｯｼｬｰ
; rung 82
LD 133.05  ; 単動:戻り
ANDNOT 13.10  ; 排出ﾓｰﾀ原点ｾﾝｻ
LD 133.06  ; 単動:排出
OR 133.07  ; 単動:払出
LD 13.10  ; 排出ﾓｰﾀ原点ｾﾝｻ
ORNOT W511.14  ; DEBUG_EM1_2nd_排出CV
ANDLD
ORLD
OUT 99.04  ; IL:排出CV_START
; rung 83
LDNOT 13.10  ; 排出ﾓｰﾀ原点ｾﾝｻ
OUT 99.05  ; IL:戻り
; rung 84
LD 13.10  ; 排出ﾓｰﾀ原点ｾﾝｻ
OR 13.11  ; 排出ﾓｰﾀ動点ｾﾝｻ
OUT 99.06  ; IL:排出
; rung 85
LD 13.10  ; 排出ﾓｰﾀ原点ｾﾝｻ
LDNOT W511.14  ; DEBUG_EM1_2nd_排出CV
ANDNOT 13.11  ; 排出ﾓｰﾀ動点ｾﾝｻ
ORLD
OUT 99.07  ; IL:払出
; rung 86
LD 60.10  ; 主軸RB_復帰終了保持
ANDNOT 1.10  ; RB:MOVE_主軸
OUT 99.08  ; IL:ﾁｬｯｸ1
; rung 87
LD 60.10  ; 主軸RB_復帰終了保持
ANDNOT 1.10  ; RB:MOVE_主軸
OUT 99.09  ; IL:ﾁｬｯｸ2
; rung 88
LD 60.10  ; 主軸RB_復帰終了保持
ANDNOT 1.10  ; RB:MOVE_主軸
OUT 99.10  ; IL:ﾁｬｯｸ3
; rung 89
LD P_On
OUT 99.11  ; IL:

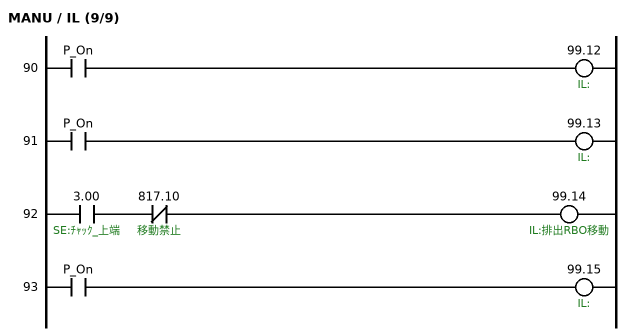
; rung 90
LD P_On
OUT 99.12  ; IL:
; rung 91
LD P_On
OUT 99.13  ; IL:
; rung 92
LD 3.00  ; SE:ﾁｬｯｸ_上端
ANDNOT 817.10  ; 移動禁止
OUT 99.14  ; IL:排出RBO移動
; rung 93
LD P_On
OUT 99.15  ; IL:

### Section TIM

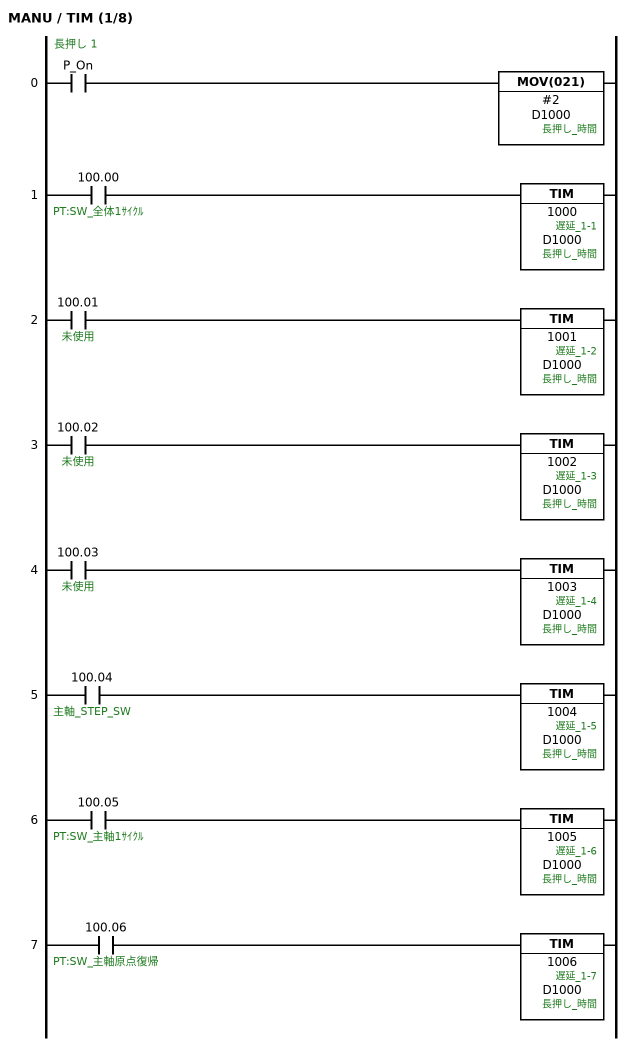
; rung 0: 長押し 1
LD P_On
MOV(021) #2 D1000  ; 長押し_時間
; rung 1
LD 100.00  ; PT:SW_全体1ｻｲｸﾙ
TIM 1000 D1000  ; 長押し_時間, 遅延_1-1
; rung 2
LD 100.01  ; 未使用
TIM 1001 D1000  ; 長押し_時間, 遅延_1-2
; rung 3
LD 100.02  ; 未使用
TIM 1002 D1000  ; 長押し_時間, 遅延_1-3
; rung 4
LD 100.03  ; 未使用
TIM 1003 D1000  ; 長押し_時間, 遅延_1-4
; rung 5
LD 100.04  ; 主軸_STEP_SW
TIM 1004 D1000  ; 長押し_時間, 遅延_1-5
; rung 6
LD 100.05  ; PT:SW_主軸1ｻｲｸﾙ
TIM 1005 D1000  ; 長押し_時間, 遅延_1-6
; rung 7
LD 100.06  ; PT:SW_主軸原点復帰
TIM 1006 D1000  ; 長押し_時間, 遅延_1-7

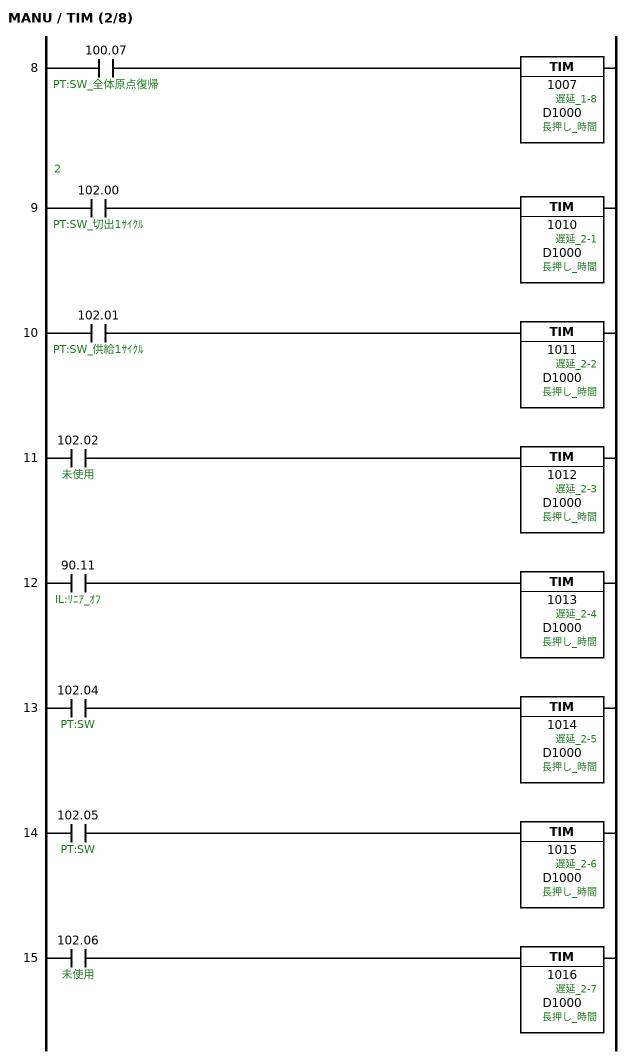
; rung 8
LD 100.07  ; PT:SW_全体原点復帰
TIM 1007 D1000  ; 長押し_時間, 遅延_1-8
; rung 9: 2
LD 102.00  ; PT:SW_切出1ｻｲｸﾙ
TIM 1010 D1000  ; 長押し_時間, 遅延_2-1
; rung 10
LD 102.01  ; PT:SW_供給1ｻｲｸﾙ
TIM 1011 D1000  ; 長押し_時間, 遅延_2-2
; rung 11
LD 102.02  ; 未使用
TIM 1012 D1000  ; 長押し_時間, 遅延_2-3
; rung 12
LD 90.11  ; IL:ﾘﾆｱ_ｵﾌ
TIM 1013 D1000  ; 長押し_時間, 遅延_2-4
; rung 13
LD 102.04  ; PT:SW
TIM 1014 D1000  ; 長押し_時間, 遅延_2-5
; rung 14
LD 102.05  ; PT:SW
TIM 1015 D1000  ; 長押し_時間, 遅延_2-6
; rung 15
LD 102.06  ; 未使用
TIM 1016 D1000  ; 長押し_時間, 遅延_2-7

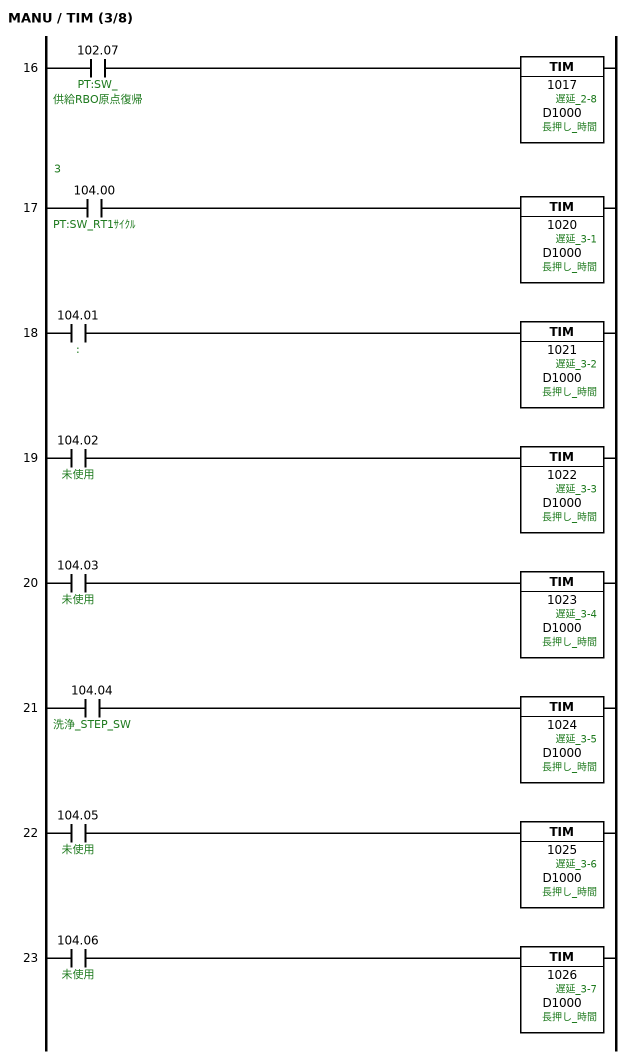
; rung 16
LD 102.07  ; PT:SW_供給RBO原点復帰
TIM 1017 D1000  ; 長押し_時間, 遅延_2-8
; rung 17: 3
LD 104.00  ; PT:SW_RT1ｻｲｸﾙ
TIM 1020 D1000  ; 長押し_時間, 遅延_3-1
; rung 18
LD 104.01  ; :
TIM 1021 D1000  ; 長押し_時間, 遅延_3-2
; rung 19
LD 104.02  ; 未使用
TIM 1022 D1000  ; 長押し_時間, 遅延_3-3
; rung 20
LD 104.03  ; 未使用
TIM 1023 D1000  ; 長押し_時間, 遅延_3-4
; rung 21
LD 104.04  ; 洗浄_STEP_SW
TIM 1024 D1000  ; 長押し_時間, 遅延_3-5
; rung 22
LD 104.05  ; 未使用
TIM 1025 D1000  ; 長押し_時間, 遅延_3-6
; rung 23
LD 104.06  ; 未使用
TIM 1026 D1000  ; 長押し_時間, 遅延_3-7

